FUNCTION _any_to_string : MaxString
VAR_INPUT
  to_transform: ANY;
END_VAR
VAR
  int_ptr: POINTER TO INT;
  real_ptr: POINTER TO REAL;
  string_ptr: POINTER TO STRING;
END_VAR

CASE UDINT_TO_INT(to_transform.TypeClass) OF
TypeClass.TYPE_INT:
  int_ptr := to_transform.pValue;
  _any_to_string := TO_STRING(int_ptr^);
TypeClass.TYPE_REAL:
  real_ptr := to_transform.pValue;
  _any_to_string := TO_STRING(real_ptr^);
TypeClass.TYPE_STRING:
  string_ptr := to_transform.pValue;
  _any_to_string := string_ptr^;
ELSE
  _any_to_string := '';
END_CASE

END_FUNCTION

(* stored: Version 1.1.0.1, ProductVersion 3.1.4022.7
   POU _any_to_string: Id {ac8c30cd-67ee-4e25-b911-ae2d14e6a975}, SpecialFunc None *)
